// TIA Portal V21 export
// export: Created 2026-07-27T22:10:58.774591Z, ExportSetting WithDefaults, DisplayName Totally Integrated Automation Portal, DisplayVersion V21, DisplayName SINAMICS Startdrive Advanced, DisplayVersion V21, DisplayName SINAMICS Startdrive G110M, G120, G120C, G120D, G120P, G115D, DisplayVersion V21, DisplayName SINAMICS Startdrive G130, G150, S120, S150, G200, G220, S200, S210, S220, Innomotics MVD, DisplayVersion V21, DisplayName STEP 7 Professional, DisplayVersion V21, DisplayName STEP 7 Safety, DisplayVersion V21, DisplayName Tech WebApplication, DisplayVersion V21, DisplayName WinCC Basic/Comfort/Advanced, DisplayVersion V21, DisplayName WinCC Professional, DisplayVersion V21, DisplayName WinCC Unified, DisplayVersion V21
FUNCTION "MOLDE_ANALOGS" : Void   // FC128, LAD
{ S7_Optimized_Access := 'TRUE' }
VERSION : 0.1
// Parâmetros da Equação da Reta
// ANALOG_IN_4a20mA: Entrada Analógica
// Y1_CONFIG: Range mínimo Sinal de Campo
// Y2_CONFIG: Range máximo Sinal de Campo
// X1_CONFIG: Range Mínimo Entrada Analógica CLP
// X2_CONFIG: Range Máximo Entrada Analógica CLP
// COMANDO: Parâmetro enviado da IHM/SCADA
// COMANDO_VALOR: Parâmetro referente à aferição do bloco
// GRANDEZA_MAX = Valor de comunicação RS485, enviado pelo inversor 
// RANGE_MIN_CADASTRADO = Valor de leitura minimo que irá aparecer no display IHM
// RANGE_MAX_CADASTRADO = Valor de leitura maximo que irá aparecer no display IHM
// 
// Comando Aferição 8888: (FQIT-01)
// Comando Limites 9999: (FQIT-01)
// stored: AutoNumber true, IsIECCheckEnabled false, SetENOAutomatically false, UDAEnableTagReadback false
BEGIN

REGION Network 1: Aferição Equipamento (FQIT-01)
   // Aferição Entrada Analógica (FQIT-01)
   // 
   // Comando:
   // 8888: Comando de Aferição (FQIT-01)
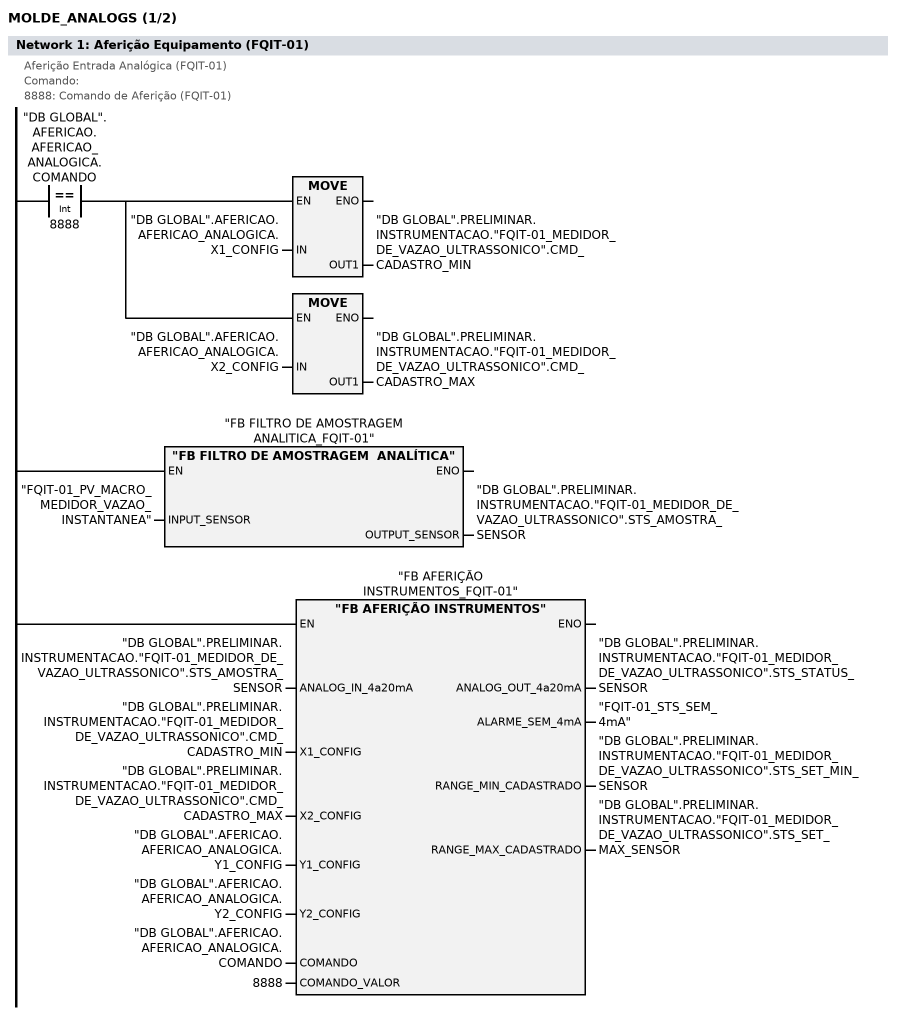
   RUNG wire#powerrail
      { S7_Templates := "SrcType := Int" } EQ_Contact(in1 := "DB GLOBAL".AFERICAO.AFERICAO_ANALOGICA.COMANDO, in2 := 8888)
      wire#w1
      Move(in := "DB GLOBAL".AFERICAO.AFERICAO_ANALOGICA.X1_CONFIG, out1 => "DB GLOBAL".PRELIMINAR.INSTRUMENTACAO."FQIT-01_MEDIDOR_DE_VAZAO_ULTRASSONICO".CMD_CADASTRO_MIN)
   END_RUNG
   RUNG wire#w1
      Move(in := "DB GLOBAL".AFERICAO.AFERICAO_ANALOGICA.X2_CONFIG, out1 => "DB GLOBAL".PRELIMINAR.INSTRUMENTACAO."FQIT-01_MEDIDOR_DE_VAZAO_ULTRASSONICO".CMD_CADASTRO_MAX)
   END_RUNG
   RUNG wire#powerrail
      "FB FILTRO DE AMOSTRAGEM  ANALITICA_FQIT-01"(INPUT_SENSOR := "FQIT-01_PV_MACRO_MEDIDOR_VAZAO_INSTANTANEA", OUTPUT_SENSOR => "DB GLOBAL".PRELIMINAR.INSTRUMENTACAO."FQIT-01_MEDIDOR_DE_VAZAO_ULTRASSONICO".STS_AMOSTRA_SENSOR)
   END_RUNG
   RUNG wire#powerrail
      "FB AFERIÇÃO INSTRUMENTOS_FQIT-01"(ANALOG_IN_4a20mA := "DB GLOBAL".PRELIMINAR.INSTRUMENTACAO."FQIT-01_MEDIDOR_DE_VAZAO_ULTRASSONICO".STS_AMOSTRA_SENSOR, X1_CONFIG := "DB GLOBAL".PRELIMINAR.INSTRUMENTACAO."FQIT-01_MEDIDOR_DE_VAZAO_ULTRASSONICO".CMD_CADASTRO_MIN, X2_CONFIG := "DB GLOBAL".PRELIMINAR.INSTRUMENTACAO."FQIT-01_MEDIDOR_DE_VAZAO_ULTRASSONICO".CMD_CADASTRO_MAX, Y1_CONFIG := "DB GLOBAL".AFERICAO.AFERICAO_ANALOGICA.Y1_CONFIG, Y2_CONFIG := "DB GLOBAL".AFERICAO.AFERICAO_ANALOGICA.Y2_CONFIG, COMANDO := "DB GLOBAL".AFERICAO.AFERICAO_ANALOGICA.COMANDO, COMANDO_VALOR := 8888, ANALOG_OUT_4a20mA => "DB GLOBAL".PRELIMINAR.INSTRUMENTACAO."FQIT-01_MEDIDOR_DE_VAZAO_ULTRASSONICO".STS_STATUS_SENSOR, ALARME_SEM_4mA => "FQIT-01_STS_SEM_4mA", RANGE_MIN_CADASTRADO => "DB GLOBAL".PRELIMINAR.INSTRUMENTACAO."FQIT-01_MEDIDOR_DE_VAZAO_ULTRASSONICO".STS_SET_MIN_SENSOR, RANGE_MAX_CADASTRADO => "DB GLOBAL".PRELIMINAR.INSTRUMENTACAO."FQIT-01_MEDIDOR_DE_VAZAO_ULTRASSONICO".STS_SET_MAX_SENSOR)
   END_RUNG
   // the same network as SCL:
   IF "DB GLOBAL".AFERICAO.AFERICAO_ANALOGICA.COMANDO = 8888 THEN
       "DB GLOBAL".PRELIMINAR.INSTRUMENTACAO."FQIT-01_MEDIDOR_DE_VAZAO_ULTRASSONICO".CMD_CADASTRO_MIN := "DB GLOBAL".AFERICAO.AFERICAO_ANALOGICA.X1_CONFIG;
       "DB GLOBAL".PRELIMINAR.INSTRUMENTACAO."FQIT-01_MEDIDOR_DE_VAZAO_ULTRASSONICO".CMD_CADASTRO_MAX := "DB GLOBAL".AFERICAO.AFERICAO_ANALOGICA.X2_CONFIG;
   END_IF;
   "FB FILTRO DE AMOSTRAGEM  ANALITICA_FQIT-01"(INPUT_SENSOR := "FQIT-01_PV_MACRO_MEDIDOR_VAZAO_INSTANTANEA",   // "FB FILTRO DE AMOSTRAGEM  ANALÍTICA"
                           OUTPUT_SENSOR => "DB GLOBAL".PRELIMINAR.INSTRUMENTACAO."FQIT-01_MEDIDOR_DE_VAZAO_ULTRASSONICO".STS_AMOSTRA_SENSOR);
   "FB AFERIÇÃO INSTRUMENTOS_FQIT-01"(ANALOG_IN_4a20mA := "DB GLOBAL".PRELIMINAR.INSTRUMENTACAO."FQIT-01_MEDIDOR_DE_VAZAO_ULTRASSONICO".STS_AMOSTRA_SENSOR,   // "FB AFERIÇÃO INSTRUMENTOS"
                           X1_CONFIG := "DB GLOBAL".PRELIMINAR.INSTRUMENTACAO."FQIT-01_MEDIDOR_DE_VAZAO_ULTRASSONICO".CMD_CADASTRO_MIN,
                           X2_CONFIG := "DB GLOBAL".PRELIMINAR.INSTRUMENTACAO."FQIT-01_MEDIDOR_DE_VAZAO_ULTRASSONICO".CMD_CADASTRO_MAX,
                           Y1_CONFIG := "DB GLOBAL".AFERICAO.AFERICAO_ANALOGICA.Y1_CONFIG,
                           Y2_CONFIG := "DB GLOBAL".AFERICAO.AFERICAO_ANALOGICA.Y2_CONFIG,
                           COMANDO := "DB GLOBAL".AFERICAO.AFERICAO_ANALOGICA.COMANDO,
                           COMANDO_VALOR := 8888,
                           ANALOG_OUT_4a20mA => "DB GLOBAL".PRELIMINAR.INSTRUMENTACAO."FQIT-01_MEDIDOR_DE_VAZAO_ULTRASSONICO".STS_STATUS_SENSOR,
                           ALARME_SEM_4mA => "FQIT-01_STS_SEM_4mA",
                           RANGE_MIN_CADASTRADO => "DB GLOBAL".PRELIMINAR.INSTRUMENTACAO."FQIT-01_MEDIDOR_DE_VAZAO_ULTRASSONICO".STS_SET_MIN_SENSOR,
                           RANGE_MAX_CADASTRADO => "DB GLOBAL".PRELIMINAR.INSTRUMENTACAO."FQIT-01_MEDIDOR_DE_VAZAO_ULTRASSONICO".STS_SET_MAX_SENSOR);
END_REGION

REGION Network 2: Limites de Operação (FQIT-01)
   // Cadastro Limites de Operação sensor (FQIT-01)
   // Alarme leitura muito baixa
   // Alarme leitura baixa
   // Alarme leitura alta
   // Alarme leitura muito alta
   // 
   // Comando:
   // 9999: Definição de Limites para (FQIT-01)
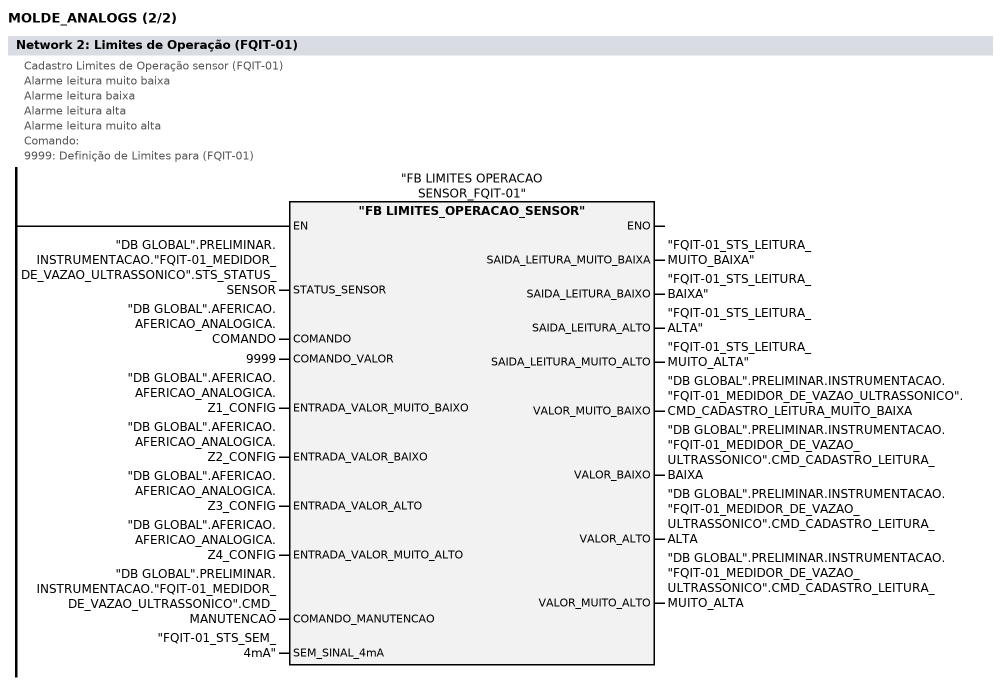
   RUNG wire#powerrail
      "FB LIMITES OPERACAO SENSOR_FQIT-01"(STATUS_SENSOR := "DB GLOBAL".PRELIMINAR.INSTRUMENTACAO."FQIT-01_MEDIDOR_DE_VAZAO_ULTRASSONICO".STS_STATUS_SENSOR, COMANDO := "DB GLOBAL".AFERICAO.AFERICAO_ANALOGICA.COMANDO, COMANDO_VALOR := 9999, ENTRADA_VALOR_MUITO_BAIXO := "DB GLOBAL".AFERICAO.AFERICAO_ANALOGICA.Z1_CONFIG, ENTRADA_VALOR_BAIXO := "DB GLOBAL".AFERICAO.AFERICAO_ANALOGICA.Z2_CONFIG, ENTRADA_VALOR_ALTO := "DB GLOBAL".AFERICAO.AFERICAO_ANALOGICA.Z3_CONFIG, ENTRADA_VALOR_MUITO_ALTO := "DB GLOBAL".AFERICAO.AFERICAO_ANALOGICA.Z4_CONFIG, COMANDO_MANUTENCAO := "DB GLOBAL".PRELIMINAR.INSTRUMENTACAO."FQIT-01_MEDIDOR_DE_VAZAO_ULTRASSONICO".CMD_MANUTENCAO, SEM_SINAL_4mA := "FQIT-01_STS_SEM_4mA", SAIDA_LEITURA_MUITO_BAIXA => "FQIT-01_STS_LEITURA_MUITO_BAIXA", SAIDA_LEITURA_BAIXO => "FQIT-01_STS_LEITURA_BAIXA", SAIDA_LEITURA_ALTO => "FQIT-01_STS_LEITURA_ALTA", SAIDA_LEITURA_MUITO_ALTO => "FQIT-01_STS_LEITURA_MUITO_ALTA", VALOR_MUITO_BAIXO => "DB GLOBAL".PRELIMINAR.INSTRUMENTACAO."FQIT-01_MEDIDOR_DE_VAZAO_ULTRASSONICO".CMD_CADASTRO_LEITURA_MUITO_BAIXA, VALOR_BAIXO => "DB GLOBAL".PRELIMINAR.INSTRUMENTACAO."FQIT-01_MEDIDOR_DE_VAZAO_ULTRASSONICO".CMD_CADASTRO_LEITURA_BAIXA, VALOR_ALTO => "DB GLOBAL".PRELIMINAR.INSTRUMENTACAO."FQIT-01_MEDIDOR_DE_VAZAO_ULTRASSONICO".CMD_CADASTRO_LEITURA_ALTA, VALOR_MUITO_ALTO => "DB GLOBAL".PRELIMINAR.INSTRUMENTACAO."FQIT-01_MEDIDOR_DE_VAZAO_ULTRASSONICO".CMD_CADASTRO_LEITURA_MUITO_ALTA)
   END_RUNG
   // the same network as SCL:
   "FB LIMITES OPERACAO SENSOR_FQIT-01"(STATUS_SENSOR := "DB GLOBAL".PRELIMINAR.INSTRUMENTACAO."FQIT-01_MEDIDOR_DE_VAZAO_ULTRASSONICO".STS_STATUS_SENSOR,   // "FB LIMITES_OPERACAO_SENSOR"
                           COMANDO := "DB GLOBAL".AFERICAO.AFERICAO_ANALOGICA.COMANDO,
                           COMANDO_VALOR := 9999,
                           ENTRADA_VALOR_MUITO_BAIXO := "DB GLOBAL".AFERICAO.AFERICAO_ANALOGICA.Z1_CONFIG,
                           ENTRADA_VALOR_BAIXO := "DB GLOBAL".AFERICAO.AFERICAO_ANALOGICA.Z2_CONFIG,
                           ENTRADA_VALOR_ALTO := "DB GLOBAL".AFERICAO.AFERICAO_ANALOGICA.Z3_CONFIG,
                           ENTRADA_VALOR_MUITO_ALTO := "DB GLOBAL".AFERICAO.AFERICAO_ANALOGICA.Z4_CONFIG,
                           COMANDO_MANUTENCAO := "DB GLOBAL".PRELIMINAR.INSTRUMENTACAO."FQIT-01_MEDIDOR_DE_VAZAO_ULTRASSONICO".CMD_MANUTENCAO,
                           SEM_SINAL_4mA := "FQIT-01_STS_SEM_4mA",
                           SAIDA_LEITURA_MUITO_BAIXA => "FQIT-01_STS_LEITURA_MUITO_BAIXA",
                           SAIDA_LEITURA_BAIXO => "FQIT-01_STS_LEITURA_BAIXA",
                           SAIDA_LEITURA_ALTO => "FQIT-01_STS_LEITURA_ALTA",
                           SAIDA_LEITURA_MUITO_ALTO => "FQIT-01_STS_LEITURA_MUITO_ALTA",
                           VALOR_MUITO_BAIXO => "DB GLOBAL".PRELIMINAR.INSTRUMENTACAO."FQIT-01_MEDIDOR_DE_VAZAO_ULTRASSONICO".CMD_CADASTRO_LEITURA_MUITO_BAIXA,
                           VALOR_BAIXO => "DB GLOBAL".PRELIMINAR.INSTRUMENTACAO."FQIT-01_MEDIDOR_DE_VAZAO_ULTRASSONICO".CMD_CADASTRO_LEITURA_BAIXA,
                           VALOR_ALTO => "DB GLOBAL".PRELIMINAR.INSTRUMENTACAO."FQIT-01_MEDIDOR_DE_VAZAO_ULTRASSONICO".CMD_CADASTRO_LEITURA_ALTA,
                           VALOR_MUITO_ALTO => "DB GLOBAL".PRELIMINAR.INSTRUMENTACAO."FQIT-01_MEDIDOR_DE_VAZAO_ULTRASSONICO".CMD_CADASTRO_LEITURA_MUITO_ALTA);
END_REGION
END_FUNCTION
